{attribute addProperty BoxType "IODEVICETYPE_ETHERCATPROT"}
{attribute addProperty Id "Beckhoff_EPP1xxxBeckhoff_EPP1xxx_AAF5AC245888736Beckhoff_EPP2xxxBeckhoff_EPP2xxx_B6CD005B168002100Beckhoff_EPP3xxxBeckhoff_EPP3xxx_F198DF1F7992999Beckhoff_EPP4xxxBeckhoff_EPP4xxx_3B08D8421312164Beckhoff_EPP5xxxBeckhoff_EPP5xxx_3599C48B1568196Beckhoff_EPP6xxxBeckhoff_EPP6xxx_9BDCB0CF5344668Beckhoff_EPP7xxxBeckhoff_EPP7xxx_834E57DE2464308Beckhoff_EPP9xxxBeckhoff_EPP9xxx_6B7D5A5F56070SyncUnitsSyncUnits_3FA29F3C21627InputsInputs_C75D3FEC1280160OutputsOutputs_47D1E803848106InfoDataInfoData_45F98C5022428"}
{attribute addProperty CRC "2373326776"}
{attribute addProperty SizeInBites "44496"}
{attribute addProperty SizeInBytes "5562"}
TYPE EtherCAT_Master_EPPxxxx_8D7617B8 :
STRUCT
	{attribute addProperty Name "Beckhoff_EPP1xxx"}
	Beckhoff_EPP1xxx : Beckhoff_EPP1xxx_AAF5AC24;
	{attribute addProperty Name "Beckhoff_EPP2xxx"}
	Beckhoff_EPP2xxx : Beckhoff_EPP2xxx_B6CD005B;
	{attribute addProperty Name "Beckhoff_EPP3xxx"}
	Beckhoff_EPP3xxx : Beckhoff_EPP3xxx_F198DF1F;
	{attribute addProperty Name "Beckhoff_EPP4xxx"}
	Beckhoff_EPP4xxx : Beckhoff_EPP4xxx_3B08D842;
	{attribute addProperty Name "Beckhoff_EPP5xxx"}
	Beckhoff_EPP5xxx : Beckhoff_EPP5xxx_3599C48B;
	{attribute addProperty Name "Beckhoff_EPP6xxx"}
	Beckhoff_EPP6xxx : Beckhoff_EPP6xxx_9BDCB0CF;
	{attribute addProperty Name "Beckhoff_EPP7xxx"}
	Beckhoff_EPP7xxx : Beckhoff_EPP7xxx_834E57DE;
	{attribute addProperty Name "Beckhoff_EPP9xxx"}
	Beckhoff_EPP9xxx : Beckhoff_EPP9xxx_6B7D5A5F;
	{attribute addProperty Name "SyncUnits"}
	SyncUnits : SyncUnits_3FA29F3C;
	{attribute addProperty Name "Inputs"}
	Inputs : Inputs_C75D3FEC;
	{attribute addProperty Name "Outputs"}
	Outputs : Outputs_47D1E803;
	{attribute addProperty Name "InfoData"}
	InfoData : InfoData_45F98C50;
END_STRUCT
END_TYPE

(* stored: Version 1.2.0.0, ProductVersion 3.1.4024.9
   DUT EtherCAT_Master_EPPxxxx_8D7617B8: Id {f28d461f-94bc-425b-b6d3-e84348bd153c} *)
